{attribute 'qualified_only'}
{attribute 'strict'}
// Düsendurchmesser in mm und die zugehärige Reduzierung des maximalen Durchflusses in mm^3/s
TYPE E_NozzleSizeFlow :
(
	fuenf 	:= 0,
	vier	:= -60,
	drei	:= -120,
	zwei 	:= -180,
	ein		:= -240
)DINT := drei;
END_TYPE

(* stored: Version 1.1.0.1
   DUT E_NozzleSizeFlow: Id {c363c4e0-eeb8-4631-8e62-dae07b6148a3} *)
